FUNCTION_BLOCK VacuumGripper EXTENDS BaseGripper
VAR_INPUT
END_VAR
VAR_OUTPUT
END_VAR
VAR
	//Hardware
	DI_TakenIn AT %I* : BOOL;
	DO_VacuumOn AT %Q* : BOOL;
	// Only used by PickAlpha
	VacuumHit AT %Q* : BOOL;
END_VAR

METHOD METH_Intake : BOOL
VAR_INPUT
END_VAR
DO_VacuumOn := TRUE;
END_METHOD

METHOD METH_Release : BOOL
VAR_INPUT
END_VAR
DO_VacuumOn := FALSE;
END_METHOD

METHOD METH_VacuumHitOff : BOOL
VAR_INPUT
END_VAR
VacuumHit := FALSE;
END_METHOD

METHOD METH_VacuumHitOn : BOOL
VAR_INPUT
END_VAR
VacuumHit := TRUE;
END_METHOD

PROPERTY WPTaken : BOOL
GET
// TODO - connect input correctly (probably hardware issue)
WPTaken := DI_TakenIn;
//WPTaken := DO_VacuumOn;
END_GET
END_PROPERTY

END_FUNCTION_BLOCK

(* stored: Version 1.1.0.1, ProductVersion 3.1.4024.4
   POU VacuumGripper: Id {fd144578-ed2c-442a-a857-49821ed88d71}, SpecialFunc None
   Method METH_Intake: Id {4637e086-4937-416b-89e4-86f1f8913a16}
   Method METH_Release: Id {f04f00e6-e3c8-441c-99c7-8ae309e0dd4e}
   Method METH_VacuumHitOff: Id {1b22ed15-b49b-4c33-a9dd-7e3bf9bed31d}
   Method METH_VacuumHitOn: Id {e06e7425-cfe1-47ee-8b03-2693e20b9ef8}
   Property WPTaken: Id {430f7e05-e654-405e-835f-733d57a19fe9}
   Get Get: Id {ef46c3b9-3d68-4550-9bc7-bef828915b28} *)
